(* IEC 61131-3 sources: POMIRTS_lab3/AS/Library_2/AsArcnet, 3 files *)

(* ---- AsArcnet.typ ---- *)
(********************************************************************
 * COPYRIGHT -- Bernecker + Rainer
 ********************************************************************
 * Library: AsArcnet
 * File: AsArcnet.typ
 * Author: B+R
 ********************************************************************
 * Data types of library AsArcnet
 ********************************************************************)

TYPE
	ARCstat_typ : 	STRUCT     (*statistic data*)
		BytesRecv : UDINT;     (*number of bytes received by Fbase*)
		BytesSend : UDINT;     (*number of bytes sent and confirmed by Fbase*)
		IntRX : UDINT;         (*receive interrupt*)
		IntTA : UDINT;         (*transmit interrupt*)
		IntENAK : UDINT;       (*excessive NAK interrupt*)
		IntNNID : UDINT;       (*new next ID interrupt*)
		IntRECON : UDINT;      (*reconfiguration interrupt*)
		ReconCnt : UDINT;      (*number of reconfigurations triggered by the nodes*)
		ErrRead : UDINT;       (*error reading from the controller*)
		ErrSend : UDINT;       (*error writing to the controller*)
		NoFreeBuf : UDINT;     (*counters for buffers are full (call ARCread as long as "status" equals ERR_OK*)
		ExcPaket : UDINT;      (*exception packet counter*)
	END_STRUCT;
END_TYPE

(* ---- AsArcnet.fun ---- *)
(********************************************************************
 * COPYRIGHT -- Bernecker + Rainer
 ********************************************************************
 * Library: AsArcnet
 * File: AsArcnet.fun
 * Author: B+R
 ********************************************************************
 * Functions and function blocks of library AsArcnet
 ********************************************************************)

FUNCTION_BLOCK ARCopen             (*opens an Arcnet device*)
	VAR_INPUT
		enable			: BOOL;    (*enables execution*)
		device			: UDINT;   (*device name given as a pointer, e.g., "SL3.SS1.IF2"*)
		mode			: UDINT;   (*initialization string given as a pointer, e.g., "/BD=1250000 /RECON=105000 /ET=2"*)
	END_VAR

	VAR_OUTPUT
		status			: UINT;    (*execution status: ERR_OK, ERR_FUB_ENABLE_FALSE, 0xXXXX = see help*)
		ident			: UDINT;   (*identifier of the opened Arcnet device*)
	END_VAR
END_FUNCTION_BLOCK

FUNCTION_BLOCK ARCclose            (*closes an Arcnet device*)
	VAR_INPUT
		enable			: BOOL;    (*enables execution*)
		ident			: UDINT;   (*identifier returned from ARCopen()*)
	END_VAR

	VAR_OUTPUT
		status			: UINT;    (*execution status: ERR_OK, ERR_FUB_ENABLE_FALSE, 0xXXXX = see help*)
	END_VAR
END_FUNCTION_BLOCK

FUNCTION_BLOCK ARCread             (*reads received frames*)
	VAR_INPUT
		enable			: BOOL;    (*enables execution*)
		ident			: UDINT;   (*identifier returned from ARCopen()*)
		buffer			: UDINT;   (*address of the receive buffer*)
		buflng			: UDINT;   (*address of the length variable of the receive buffer*)
	END_VAR

	VAR_OUTPUT
		status			: UINT;    (*execution status: ERR_OK, ERR_FUB_ENABLE_FALSE, 0xXXXX = see help*)
		node_id			: USINT;   (*identifier of the sender*)
	END_VAR
END_FUNCTION_BLOCK

FUNCTION_BLOCK ARCwrite            (*sends a frame to a receiving station*)
	VAR_INPUT
		enable			: BOOL;    (*enables execution*)
		ident			: UDINT;   (*identifier returned from ARCopen()*)
		buffer			: UDINT;   (*address of the buffer containing send data*)
		buflng			: UDINT;   (*address of the length variable of the send data*)
		node_id			: USINT;   (*identifier of the receiver*)
	END_VAR

	VAR_OUTPUT
		status			: UINT;    (*execution status: ERR_OK, ERR_FUB_ENABLE_FALSE, 0xXXXX = see help*)
	END_VAR
END_FUNCTION_BLOCK

FUNCTION_BLOCK ARCexcep            (*inserts an exception task which is called when a frame with a specified ID has been received*)
	VAR_INPUT
		enable			: BOOL;    (*enables execution*)
		ident			: UDINT;   (*identifier returned from ARCopen()*)
		node_id			: USINT;   (*identifier which triggers the exception task*)
		exc_nr			: USINT;   (*number of the exception task*)
	END_VAR

	VAR_OUTPUT
		status			: UINT;    (*execution status: ERR_OK, ERR_FUB_ENABLE_FALSE, 0xXXXX = see help*)
	END_VAR
END_FUNCTION_BLOCK

FUNCTION_BLOCK ARCinfo             (*reads various information about FbArcnet*)
	VAR_INPUT
		enable			: BOOL;    (*enables execution*)
		ident			: UDINT;   (*identifier returned from ARCopen()*)
	END_VAR

	VAR_OUTPUT
		status			: UINT;    (*execution status: ERR_OK, ERR_FUB_ENABLE_FALSE, 0xXXXX = see help*)
		node_id			: USINT;   (*particular node number set on the hardware switch*)
		statadr			: UDINT;   (*address of the statistic variables of type ARCstat_typ_structure*)
	END_VAR
END_FUNCTION_BLOCK

FUNCTION_BLOCK ARCxread            (*reads received frames from an exception task*)
	VAR_INPUT
		enable			: BOOL;    (*enables execution*)
		ident			: UDINT;   (*identifier returned from ARCopen()*)
		buffer			: UDINT;   (*address of the receive buffer*)
		buflng			: UDINT;   (*address of the length variable of the receive buffer*)
	END_VAR

	VAR_OUTPUT
		status			: UINT;    (*execution status: ERR_OK, ERR_FUB_ENABLE_FALSE, 0xXXXX = see help*)
		node_id			: USINT;   (*identifier of the sender*)
	END_VAR
END_FUNCTION_BLOCK

(* ---- AsArcnet.var ---- *)
(********************************************************************
 * COPYRIGHT -- Bernecker + Rainer
 ********************************************************************
 * Library: AsArcnet
 * File: AsArcnet.var
 * Author: B+R
 ********************************************************************
 * Local variables of library AsArcnet
 ********************************************************************)

VAR CONSTANT
	ERR_ARCLIB_BUFLNG 				: UINT 		:= 27905;    (*specified buffer length invalid*)
	ERR_ARCLIB_DEVICE 				: UINT		:= 27903;    (*specified device invalid*)
	ERR_ARCLIB_FBASE  				: UINT		:= 27907;    (*internal FBASE error*)
	ERR_ARCLIB_INIT_UP 				: UINT		:= 27909;    (*init-SP calls not yet supported*)
	ERR_ARCLIB_INVALID_IDENT 		: UINT		:= 27901;    (*specified identifier invalid*)
	ERR_ARCLIB_INVALID_NODEID 		: UINT		:= 27908;    (*specified node identifier invalid*)
	ERR_ARCLIB_INVALID_PARAM 		: UINT		:= 27904;    (*specified parameters invalid*)
	ERR_ARCLIB_NO_FRAME 			: UINT		:= 27906;    (*no data received*)
	ERR_ARCLIB_NO_MORE_IDENTS 		: UINT		:= 27902;    (*no more identifiers available*)
	ERR_ARCLIB_QUEUE 				: UINT		:= 27900;    (*error in asynchronous operation*)
	ERR_ARCLIB_RECV_BUSY 			: UINT		:= 27910;    (*receiver busy*)
	ERR_ARCLIB_SEND_ACTIV 			: UINT		:= 27911;    (*sender active*)
END_VAR
